FUNCTION_BLOCK FB_EL4024
VAR_INPUT PERSISTENT

	deviceConfig    : EL4024_DEV_CONFIG; // Configuration settings for the CT121F device
	
END_VAR
VAR_INPUT
		
	Channel1  : REAL;
	Channel2  : REAL;
	Channel3  : REAL;
	Channel4  : REAL;
	
END_VAR
VAR
	    PDOS : EL4024_PDOS; // Process Data Objects for RWPT01D communication
END_VAR

_AnalogOutputs();

METHOD PRIVATE _AnalogOutputs
VAR_INPUT
END_VAR
// Calculate the actual motor speed
PDOS.HwToPLC.Channel1 := REAL_TO_INT(_Scale(
    X	 := Channel1, 
    I_LO := deviceConfig.channel1InputLow, 
    I_HI := deviceConfig.channel1InputHigh, 
    O_LO := deviceConfig.channel1OutputLow, 
    O_HI := deviceConfig.channel1OutputHigh
));
// Calculate the actual motor speed
PDOS.HwToPLC.Channel2 := REAL_TO_INT(_Scale(
    X	 := Channel2, 
    I_LO := deviceConfig.channel2InputLow, 
    I_HI := deviceConfig.channel2InputHigh, 
    O_LO := deviceConfig.channel2OutputLow, 
    O_HI := deviceConfig.channel2OutputHigh
));
// Calculate the actual motor speed
PDOS.HwToPLC.Channel3 := REAL_TO_INT(_Scale(
    X	 := Channel3, 
    I_LO := deviceConfig.channel3InputLow, 
    I_HI := deviceConfig.channel3InputHigh, 
    O_LO := deviceConfig.channel3OutputLow, 
    O_HI := deviceConfig.channel3OutputHigh
));
// Calculate the actual motor speed
PDOS.HwToPLC.Channel4 := REAL_TO_INT(_Scale(
    X	 := Channel4, 
    I_LO := deviceConfig.channel4InputLow, 
    I_HI := deviceConfig.channel4InputHigh, 
    O_LO := deviceConfig.channel4OutputLow, 
    O_HI := deviceConfig.channel4OutputHigh
));
END_METHOD

METHOD PRIVATE _Scale : REAL
VAR_INPUT
	
	X : REAL;
	I_LO : REAL;
	I_HI : REAL;
	O_LO : REAL;
	O_HI : REAL;
	
END_VAR
IF I_LO = I_HI THEN
	_Scale := O_LO;
ELSE
	_Scale := (O_HI - O_LO) / (I_HI - I_LO) * (LIMIT(I_LO, X, I_HI) - I_LO) + O_LO;
END_IF;
END_METHOD

END_FUNCTION_BLOCK

(* stored: Version 1.1.0.1, ProductVersion 3.1.4024.15
   POU FB_EL4024: Id {02396d91-213e-45d3-ac55-3cebee6a1740}, SpecialFunc None
   Method _AnalogOutputs: Id {b6c74ff4-14ae-430a-a566-8906bd2e1ef7}
   Method _Scale: Id {3ae275fb-aea2-488b-865f-00cc3fe6849b} *)
